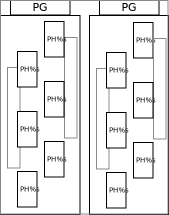
VISUALIZATION _VISU_PmEnable  // 169x215
VAR_IN_OUT
  mInst : FB_PrintModule_Base;
END_VAR
    RoundedRectangle (0,15 80x200), tooltip "WorkerPrint enable"
        toggle mInst.fbWorkerPrint[2]._bEnable
    Frame (64,37 13x101)
        shows _VISU_PcMiniVertical(m_Inst := mInst._pPc[3]^)
    Frame (7,67 13x101)
        shows _VISU_PcMiniVertical(m_Inst := mInst._pPc[4]^)
    RoundedRectangle (89,15 80x200), tooltip "WorkerPrint enable"
        toggle mInst.fbWorkerPrint[1]._bEnable
    Rectangle (133,22 20x36)
        toggle mInst._pPh[1]^._pAdsIf^.bI_Enable
    Rectangle (125,30 36x20), angle 270, "PH%s", tooltip "%s", text variable: mInst._pPh[1]^._lIdx
        p4168582468: mInst._pPh[1]^._pAdsIf^.aO_Name
    Frame (153,38 13x101), tooltip "%s"
        shows _VISU_PcMiniVertical(m_Inst := mInst._pPc[1]^)
    Frame (96,68 13x101)
        shows _VISU_PcMiniVertical(m_Inst := mInst._pPc[2]^)
    Rectangle (133,82 20x36)
        toggle mInst._pPh[2]^._pAdsIf^.bI_Enable
    Rectangle (133,142 20x36)
        toggle mInst._pPh[3]^._pAdsIf^.bI_Enable
    Rectangle (106,52 20x36)
        toggle mInst._pPh[4]^._pAdsIf^.bI_Enable
    Rectangle (106,112 20x36)
        toggle mInst._pPh[5]^._pAdsIf^.bI_Enable
    Rectangle (106,172 20x36)
        toggle mInst._pPh[6]^._pAdsIf^.bI_Enable
    Rectangle (125,90 36x20), angle 270, "PH%s", tooltip "%s", text variable: mInst._pPh[2]^._lIdx
        p4168582468: mInst._pPh[2]^._pAdsIf^.aO_Name
    Rectangle (125,150 36x20), angle 270, "PH%s", tooltip "%s", text variable: mInst._pPh[3]^._lIdx
        p4168582468: mInst._pPh[3]^._pAdsIf^.aO_Name
    Rectangle (98,60 36x20), angle 270, "PH%s", tooltip "%s", text variable: mInst._pPh[4]^._lIdx
        p4168582468: mInst._pPh[4]^._pAdsIf^.aO_Name
    Rectangle (98,120 36x20), angle 270, "PH%s", tooltip "%s", text variable: mInst._pPh[5]^._lIdx
        p4168582468: mInst._pPh[5]^._pAdsIf^.aO_Name
    Rectangle (98,180 36x20), angle 270, "PH%s", tooltip "%s", text variable: mInst._pPh[6]^._lIdx
        p4168582468: mInst._pPh[6]^._pAdsIf^.aO_Name
    Rectangle (44,21 20x36)
        toggle mInst._pPh[7]^._pAdsIf^.bI_Enable
    Rectangle (36,29 36x20), angle 270, "PH%s", tooltip "%s", text variable: mInst._pPh[7]^._lIdx
        p4168582468: mInst._pPh[7]^._pAdsIf^.aO_Name
    Rectangle (44,81 20x36)
        toggle mInst._pPh[8]^._pAdsIf^.bI_Enable
    Rectangle (44,141 20x36)
        toggle mInst._pPh[9]^._pAdsIf^.bI_Enable
    Rectangle (17,51 20x36)
        toggle mInst._pPh[10]^._pAdsIf^.bI_Enable
    Rectangle (17,111 20x36)
        toggle mInst._pPh[11]^._pAdsIf^.bI_Enable
    Rectangle (17,171 20x36)
        toggle mInst._pPh[12]^._pAdsIf^.bI_Enable
    Rectangle (36,89 36x20), angle 270, "PH%s", tooltip "%s", text variable: mInst._pPh[8]^._lIdx
        p4168582468: mInst._pPh[8]^._pAdsIf^.aO_Name
    Rectangle (36,149 36x20), angle 270, "PH%s", tooltip "%s", text variable: mInst._pPh[9]^._lIdx
        p4168582468: mInst._pPh[9]^._pAdsIf^.aO_Name
    Rectangle (9,59 36x20), angle 270, "PH%s", tooltip "%s", text variable: mInst._pPh[10]^._lIdx
        p4168582468: mInst._pPh[10]^._pAdsIf^.aO_Name
    Rectangle (9,119 36x20), angle 270, "PH%s", tooltip "%s", text variable: mInst._pPh[11]^._lIdx
        p4168582468: mInst._pPh[11]^._pAdsIf^.aO_Name
    Rectangle (9,179 36x20), angle 270, "PH%s", tooltip "%s", text variable: mInst._pPh[12]^._lIdx
        p4168582468: mInst._pPh[12]^._pAdsIf^.aO_Name
    RoundedRectangle (99,0 60x15), "PG", tooltip "PG enable"
        toggle mInst.fbWorkerPrint[1]._pAdsPg^.bI_Enable
    RoundedRectangle (10,0 60x15), "PG", tooltip "PG Enable"
        toggle mInst.fbWorkerPrint[2]._pAdsPg^.bI_Enable
END_VISUALIZATION

(* stored: Version 1.1.0.1, ProductVersion 3.1.4024.11
   Visu _VISU_PmEnable: Id {d729b797-a6c2-45a8-b0bb-a221c2872dd1} *)
